// TIA Portal V20 export
// export: Created 2025-12-01T14:57:45.3034837Z, ExportSetting None, DisplayName Totally Integrated Automation Portal, DisplayVersion V20 Update 3, DisplayName TIA Portal Openness, DisplayVersion V20 Update 3, DisplayName TIA Portal Version Control Interface, DisplayVersion V20 Update 3, DisplayName STEP 7 Professional, DisplayVersion V20 Update 3, DisplayName STEP 7 Safety, DisplayVersion V20 Update 2, DisplayName WinCC Basic/Comfort/Advanced, DisplayVersion V20 Update 3, DisplayName WinCC Professional, DisplayVersion V20 Update 3, DisplayName WinCC Unified, DisplayVersion V20 Update 3
FUNCTION "FC789_Tratamiento_mensajes_Router" : Void   // FC789, LAD
{ S7_Optimized_Access := 'FALSE' }
// stored: AutoNumber false, SetENOAutomatically false
   VAR_TEMP
      separador : Char;
      final : Char;
      ESPACIO : Char;
      retval_split : Int;
      retval : Int;
      posicion_split : UDInt;
      modo_split : DWord;
      numero_mensajes : Int;
      contador : Int;
      tamaño : Int;
      EVENTO_MENSAJE : String[4];
   END_VAR
   VAR_TEMP   // added for the SCL form of the ladder/FBD networks
      _w1 : Bool;
      _w2 : Bool;
   END_VAR
BEGIN

REGION Network 1 (SCL): inicialización
   REGION inicialiacion
       #final := ' ';
       #separador := ';';
       #modo_split := 0;
       #modo_split.%X0 := false;
       #modo_split.%X1 := true;
       #modo_split.%X3 := FALSE;
       #modo_split.%X4 := true;
       #posicion_split := 0;
       #ESPACIO := ' ';
       #numero_mensajes := 0;

       // evaluo si hay algun mensaje que impida que pueda realizar la segmentación del nuevo bloque
       // 
      #tamaño:= LEN("DB199_eventos_convertidos".evento[0]);

   END_REGION
END_REGION

REGION Network 2
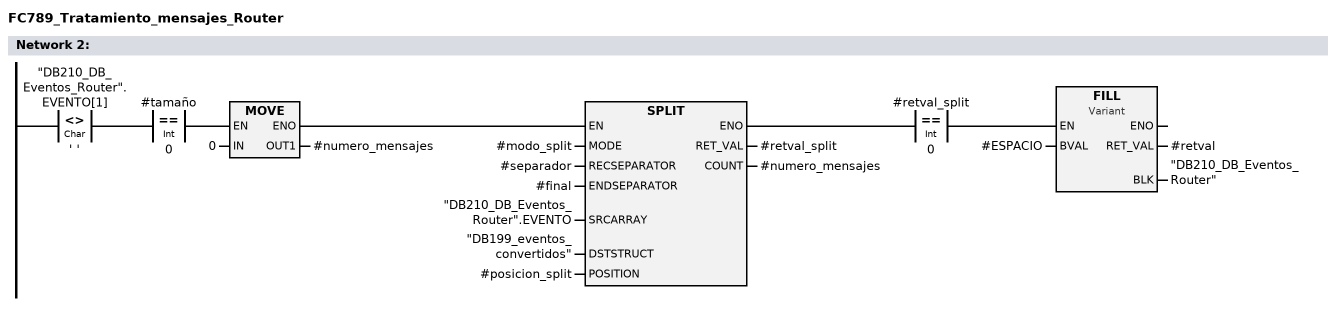
   RUNG wire#powerrail
      { S7_Templates := "SrcType := Char" } NE_Contact(in1 := "DB210_DB_Eventos_Router".EVENTO[1], in2 := ' ')
      { S7_Templates := "SrcType := Int" } EQ_Contact(in1 := #tamaño, in2 := 0)
      Move(in := 0, out1 => #numero_mensajes)
      SPLIT(Mode := #modo_split, RecSeparator := #separador, EndSeparator := #final, SrcArray := "DB210_DB_Eventos_Router".EVENTO, DstStruct := "DB199_eventos_convertidos", Position := #posicion_split, Ret_Val => #retval_split, Count => #numero_mensajes)
      { S7_Templates := "SrcType := Int" } EQ_Contact(in1 := #retval_split, in2 := 0)
      { S7_Templates := "ptr_type := Variant" } FILL(BVAL := #ESPACIO, RET_VAL => #retval, BLK => "DB210_DB_Eventos_Router")
   END_RUNG
   // the same network as SCL:
   #_w1 := ("DB210_DB_Eventos_Router".EVENTO[1] <> ' ') AND (#tamaño = 0);
   IF #_w1 THEN #numero_mensajes := 0; END_IF;
   #retval_split := SPLIT(EN := #_w1,
                          Mode := #modo_split,
                          RecSeparator := #separador,
                          EndSeparator := #final,
                          SrcArray := "DB210_DB_Eventos_Router".EVENTO,
                          DstStruct := "DB199_eventos_convertidos",
                          Position := #posicion_split,
                          Count => #numero_mensajes,
                          ENO => #_w2);
   IF #_w2 AND (#retval_split = 0) THEN
       #retval := FILL(BVAL := #ESPACIO, BLK => "DB210_DB_Eventos_Router");
   END_IF;
END_REGION

REGION Network 3 (SCL): Bucle que recorre mensajes
   IF #numero_mensajes>0 THEN
       FOR #contador := 0 TO #numero_mensajes  BY 1 DO

           // voy a tener en cuenta que los cuatro primeros caracteres del string convertido siempre van a ser el tipo de mensaje que tengo que tratar
           // 
           #EVENTO_MENSAJE := LEFT(IN := "DB199_eventos_convertidos".evento[#contador], L := 4);

           REGION Evento_RUES
               IF #EVENTO_MENSAJE = 'RUES' THEN
                   // GENERO UNA RUTA DE ELTIQUETA ESPECIAL
                   "FC782_Evento_RUES"(#contador);
                   "DB199_eventos_convertidos".evento[#contador] := DELETE(IN := "DB199_eventos_convertidos".evento[#contador], L := 0, P := 0);
                   #numero_mensajes -= 1;
                   CONTINUE;
               END_IF;
           END_REGION

           REGION Evento_RUET
               IF #EVENTO_MENSAJE = 'RUET' THEN
                   "FC780_Evento_RUET"(#contador);

                   "DB199_eventos_convertidos".evento[#contador] := DELETE(IN := "DB199_eventos_convertidos".evento[#contador], L := 0, P := 0);
                   #numero_mensajes -= 1;
                   CONTINUE;
           END_IF;
           END_REGION

           REGION Evento_BOET
               IF #EVENTO_MENSAJE = 'BOET' THEN
                   // ELIMINO UNA ETIQUETA DE LA BBDD

                   "FC783_Evento_BOET"(#contador);
                   "DB199_eventos_convertidos".evento[#contador] := DELETE(IN := "DB199_eventos_convertidos".evento[#contador], L := 0, P := 0);
                   #numero_mensajes -= 1;
                   CONTINUE;
               END_IF;
           END_REGION

           REGION Evento_BOBD
               IF #EVENTO_MENSAJE = 'BOBD' THEN
                   // BORRO LA BBDD   
                   "FC900_Reset_DB_Offset"(DB_A_RESET := "DB212_Cola_Activa",
                                           BORRAR_DESTE_BYTE := 0);
                   "FC900_Reset_DB_Offset"(DB_A_RESET := "DB201_RegEtiquetas_0001_1000",
                                           BORRAR_DESTE_BYTE := 0);
                   "FC900_Reset_DB_Offset"(DB_A_RESET := "DB202_RegEtiquetas_1001_2000",
                                           BORRAR_DESTE_BYTE := 0);
                   "FC900_Reset_DB_Offset"(DB_A_RESET := "DB203_RegEtiquetas_2001_3000",
                                           BORRAR_DESTE_BYTE := 0);
                   "FC900_Reset_DB_Offset"(DB_A_RESET := "DB204_RegEtiquetas_3001_4000",
                                           BORRAR_DESTE_BYTE := 0);
                   "FC900_Reset_DB_Offset"(DB_A_RESET := "DB209_Reg_Etquetas_Esp_Activa",
                                           BORRAR_DESTE_BYTE := 0);
                   // supervisión de los mensajes tratados. borrar luego
                   // 

                   // borrado del evento que ya hemos tratado
                   "DB199_eventos_convertidos".evento[#contador] := DELETE(IN := "DB199_eventos_convertidos".evento[#contador], L := 0, P := 0);
                   #numero_mensajes -= 1;
                   CONTINUE;
               END_IF;
           END_REGION
           REGION Evento_ORDE
               IF #EVENTO_MENSAJE = 'ORDE' THEN
                   // MENSAJE ORDE EN MESA

                   "FC781_Evento_ORDE"(#contador);
                   "DB199_eventos_convertidos".evento[#contador] := DELETE(IN := "DB199_eventos_convertidos".evento[#contador], L := 0, P := 0);
                   #numero_mensajes -= 1;
                   CONTINUE;
               END_IF;
           END_REGION
           REGION Evento_INIR
               IF #EVENTO_MENSAJE = 'INIR' THEN
                   //MENSAJE DE INCIALIZACION

                   "FC784_Evento_INIR"(#contador);
                   "DB199_eventos_convertidos".evento[#contador] := DELETE(IN := "DB199_eventos_convertidos".evento[#contador], L := 0, P := 0);
                   #numero_mensajes -= 1;
                   CONTINUE;
               END_IF;
           END_REGION

           // Statement section FOR

       END_FOR;

   END_IF;
END_REGION
END_FUNCTION
